% RSLogix 500 project 01. Basic_Instructions.RSS, saved by version 8.30.00.16 %
PROJECT "UNTITLED"    % processor: Bul.1763 MicroLogix 1100 Series B %

PROGRAM FILES
  LAD 2 "MAIN"  8 rungs
  LAD 3 "RTO E RES"  4 rungs
  LAD 4 "NEG E ABS"  3 rungs
  LAD 5 "RET E TND"  6 rungs
  LAD 6 "SUB RET"  6 rungs
  LAD 7 "AND, OR"  7 rungs  % And, Or, Not, Clear %
  LAD 8 "AIC E ACI"  9 rungs
  LAD 9 "AEC E AEX"  5 rungs
  LAD 10 "ACN E ASR"  5 rungs

DATA FILES
  O0 OUTPUT  4 elements
  I1 INPUT  6 elements
  S2 STATUS  66 elements
  B3 BINARY  2 elements
  T4 TIMER  2 elements
  C5 COUNTER  1 elements
  R6 CONTROL  1 elements
  N7 INTEGER  6 elements
  F8 FLOAT  1 elements
  B9 BINARY  6 elements
  ST10 STRINGS  12 elements
  N11 INTEIROS  15 elements

LADDER 2 "MAIN"
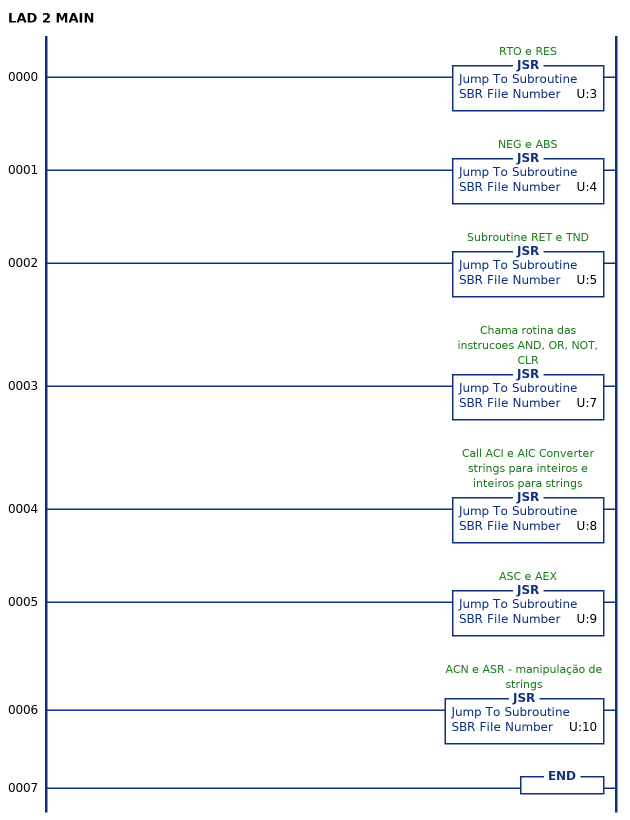
% Rung: 0 %
SOR JSR U:3 EOR
%   U:3  "RTO e RES" %
% Rung: 1 %
SOR JSR U:4 EOR
%   U:4  "NEG e ABS" %
% Rung: 2 %
SOR JSR U:5 EOR
%   U:5  "Subroutine RET e TND" %
% Rung: 3 %
SOR JSR U:7 EOR
%   U:7  "Chama rotina das instrucoes AND, OR, NOT, CLR" %
% Rung: 4 %
SOR JSR U:8 EOR
%   U:8  "Call ACI e AIC Converter strings para inteiros e inteiros para strings" %
% Rung: 5 %
SOR JSR U:9 EOR
%   U:9  "ASC e AEX" %
% Rung: 6 %
SOR JSR U:10 EOR
%   U:10  "ACN e ASR - manipulação de strings" %
% Rung: 7 %
SOR END EOR

LADDER 3 "RTO E RES"
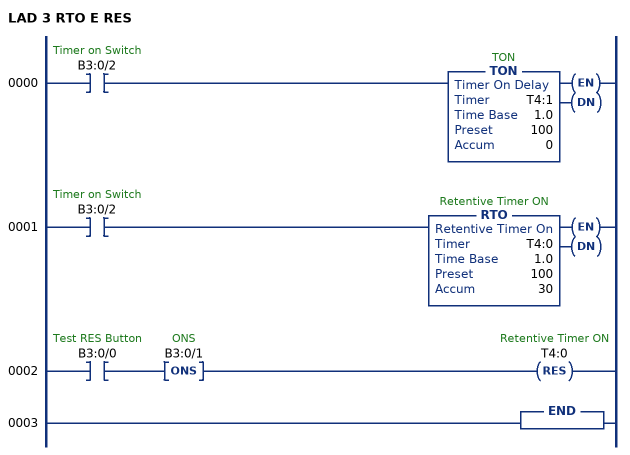
% Rung: 0 %
SOR XIC B3:0/2 TON T4:1 1.0 100 0 EOR
%   B3:0/2  "Timer on Switch" %
%   T4:1  "TON" %
% Rung: 1 %
SOR XIC B3:0/2 RTO T4:0 1.0 100 30 EOR
%   B3:0/2  "Timer on Switch" %
%   T4:0  "Retentive Timer ON" %
% Rung: 2 %
SOR XIC B3:0/0 ONS B3:0/1 RES T4:0 EOR
%   B3:0/0  "Test RES Button" %
%   B3:0/1  "ONS" %
%   T4:0  "Retentive Timer ON" %
% Rung: 3 %
SOR END EOR

LADDER 4 "NEG E ABS"
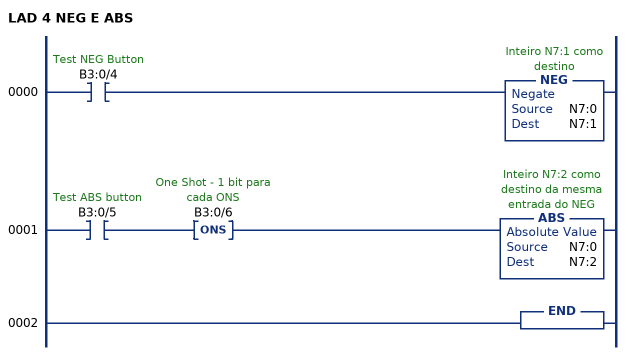
% Rung: 0 %
SOR XIC B3:0/4 NEG N7:0 N7:1 EOR
%   B3:0/4  "Test NEG Button" %
%   N7:0  "Inteiro N7:0 como entrada" %
%   N7:1  "Inteiro N7:1 como destino" %
% Rung: 1 %
SOR XIC B3:0/5 ONS B3:0/6 ABS N7:0 N7:2 EOR
%   B3:0/5  "Test ABS button" %
%   B3:0/6  "One Shot - 1 bit para cada ONS" %
%   N7:0  "Inteiro N7:0 como entrada" %
%   N7:2  "Inteiro N7:2 como destino da mesma entrada do NEG" %
% Rung: 2 %
SOR END EOR

LADDER 5 "RET E TND"
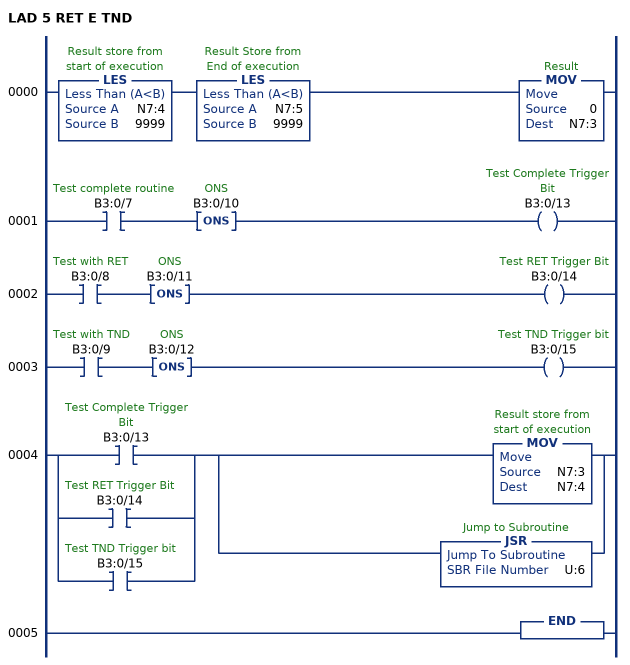
% Rung: 0 %
SOR LES N7:4 9999 LES N7:5 9999 MOV 0 N7:3 EOR
%   N7:4  "Result store from start of execution" %
%   N7:5  "Result Store from End of execution" %
%   N7:3  "Result" %
% Rung: 1 %
SOR XIC B3:0/7 ONS B3:0/10 OTE B3:0/13 EOR
%   B3:0/7  "Test complete routine" %
%   B3:0/10  "ONS" %
%   B3:0/13  "Test Complete Trigger Bit" %
% Rung: 2 %
SOR XIC B3:0/8 ONS B3:0/11 OTE B3:0/14 EOR
%   B3:0/8  "Test with RET" %
%   B3:0/11  "ONS" %
%   B3:0/14  "Test RET Trigger Bit" %
% Rung: 3 %
SOR XIC B3:0/9 ONS B3:0/12 OTE B3:0/15 EOR
%   B3:0/9  "Test with TND" %
%   B3:0/12  "ONS" %
%   B3:0/15  "Test TND Trigger bit" %
% Rung: 4 %
SOR BST XIC B3:0/13 NXB XIC B3:0/14 NXB XIC B3:0/15 BND BST MOV N7:3 N7:4 NXB JSR U:6 BND EOR
%   B3:0/13  "Test Complete Trigger Bit" %
%   B3:0/14  "Test RET Trigger Bit" %
%   B3:0/15  "Test TND Trigger bit" %
%   N7:3  "Result" %
%   N7:4  "Result store from start of execution" %
%   U:6  "Jump to Subroutine" %
% Rung: 5 %
SOR END EOR

LADDER 6 "SUB RET"
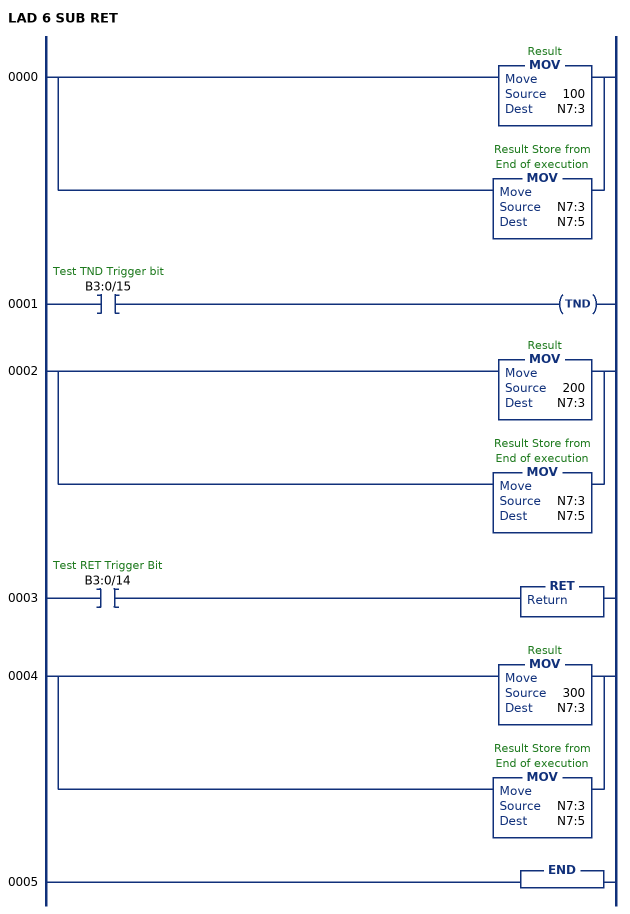
% Rung: 0 %
SOR BST MOV 100 N7:3 NXB MOV N7:3 N7:5 BND EOR
%   N7:3  "Result" %
%   N7:5  "Result Store from End of execution" %
% Rung: 1 %
SOR XIC B3:0/15 TND EOR
%   B3:0/15  "Test TND Trigger bit" %
% Rung: 2 %
SOR BST MOV 200 N7:3 NXB MOV N7:3 N7:5 BND EOR
%   N7:3  "Result" %
%   N7:5  "Result Store from End of execution" %
% Rung: 3 %
SOR XIC B3:0/14 RET EOR
%   B3:0/14  "Test RET Trigger Bit" %
% Rung: 4 %
SOR BST MOV 300 N7:3 NXB MOV N7:3 N7:5 BND EOR
%   N7:3  "Result" %
%   N7:5  "Result Store from End of execution" %
% Rung: 5 %
SOR END EOR

LADDER 7 "AND, OR"    % And, Or, Not, Clear %
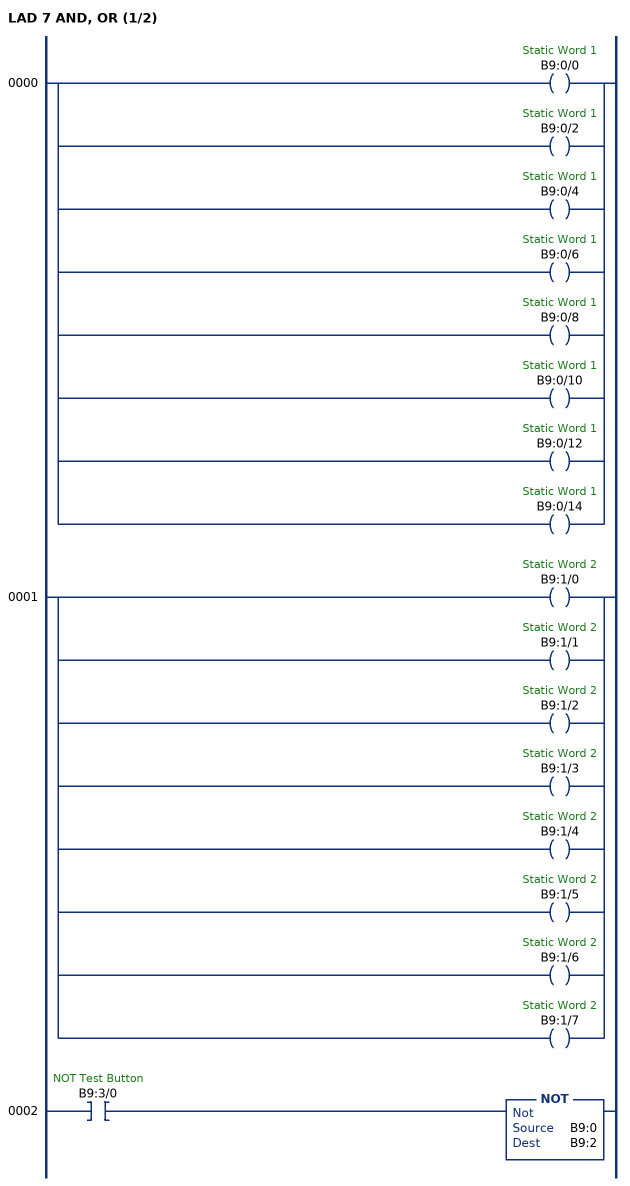
% Rung: 0 %
SOR BST OTE B9:0/0 NXB OTE B9:0/2 NXB OTE B9:0/4 NXB OTE B9:0/6 NXB OTE B9:0/8 NXB OTE B9:0/10 NXB OTE B9:0/12 NXB OTE B9:0/14 BND EOR
%   B9:0/0  "Static Word 1" %
%   B9:0/2  "Static Word 1" %
%   B9:0/4  "Static Word 1" %
%   B9:0/6  "Static Word 1" %
%   B9:0/8  "Static Word 1" %
%   B9:0/10  "Static Word 1" %
%   B9:0/12  "Static Word 1" %
%   B9:0/14  "Static Word 1" %
% Rung: 1 %
SOR BST OTE B9:1/0 NXB OTE B9:1/1 NXB OTE B9:1/2 NXB OTE B9:1/3 NXB OTE B9:1/4 NXB OTE B9:1/5 NXB OTE B9:1/6 NXB OTE B9:1/7 BND EOR
%   B9:1/0  "Static Word 2" %
%   B9:1/1  "Static Word 2" %
%   B9:1/2  "Static Word 2" %
%   B9:1/3  "Static Word 2" %
%   B9:1/4  "Static Word 2" %
%   B9:1/5  "Static Word 2" %
%   B9:1/6  "Static Word 2" %
%   B9:1/7  "Static Word 2" %
% Rung: 2 %
SOR XIC B9:3/0 NOT B9:0 B9:2 EOR
%   B9:3/0  "NOT Test Button" %
%   B9:0  "Result Word" %

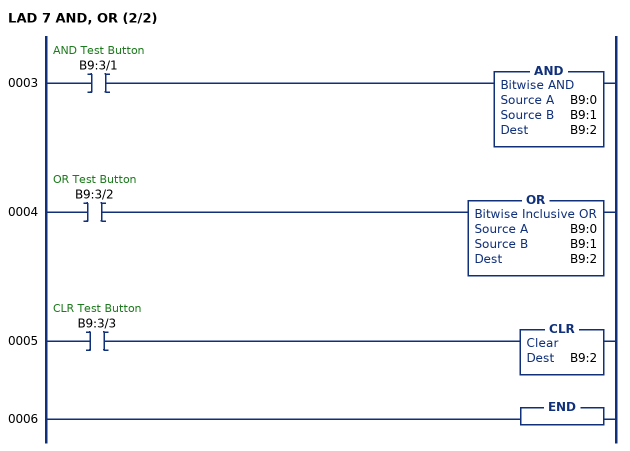
% Rung: 3 %
SOR XIC B9:3/1 AND B9:0 B9:1 B9:2 EOR
%   B9:3/1  "AND Test Button" %
%   B9:0  "Result Word" %
%   B9:1  "Result Word" %
% Rung: 4 %
SOR XIC B9:3/2 OR B9:0 B9:1 B9:2 EOR
%   B9:3/2  "OR Test Button" %
%   B9:0  "Result Word" %
%   B9:1  "Result Word" %
% Rung: 5 %
SOR XIC B9:3/3 CLR B9:2 EOR
%   B9:3/3  "CLR Test Button" %
% Rung: 6 %
SOR END EOR

LADDER 8 "AIC E ACI"
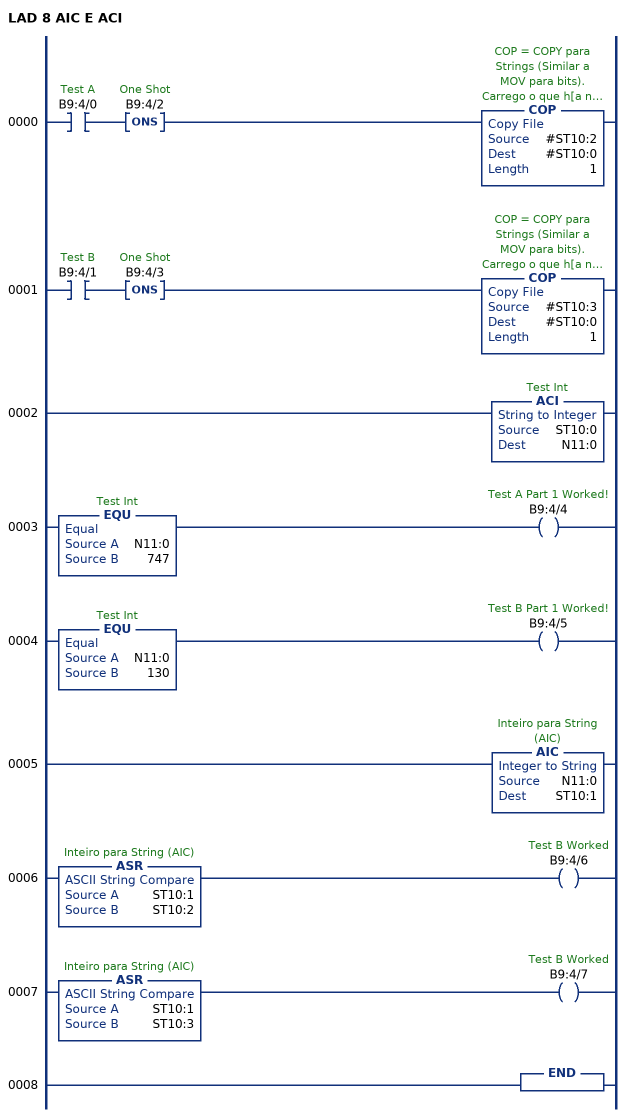
% Rung: 0 %
SOR XIC B9:4/0 ONS B9:4/2 COP #ST10:2 #ST10:0 1 EOR
%   B9:4/0  "Test A" %
%   B9:4/2  "One Shot" %
%   ST10:2  "COP = COPY para Strings. Carrego o valor da String ST9:2 para ST9:0" %
%   ST10:0  "COP = COPY para Strings (Similar a MOV para bits). Carrego o que h[a na String ST10:2 0" %
% Rung: 1 %
SOR XIC B9:4/1 ONS B9:4/3 COP #ST10:3 #ST10:0 1 EOR
%   B9:4/1  "Test B" %
%   B9:4/3  "One Shot" %
%   ST10:3  "Test String" %
%   ST10:0  "COP = COPY para Strings (Similar a MOV para bits). Carrego o que h[a na String ST10:2 0" %
% Rung: 2 %
SOR ACI ST10:0 N11:0 EOR
%   ST10:0  "COP = COPY para Strings (Similar a MOV para bits). Carrego o que h[a na String ST10:2 0" %
%   N11:0  "Test Int" %
% Rung: 3 %
SOR EQU N11:0 747 OTE B9:4/4 EOR
%   N11:0  "Test Int" %
%   B9:4/4  "Test A Part 1 Worked!" %
% Rung: 4 %
SOR EQU N11:0 130 OTE B9:4/5 EOR
%   N11:0  "Test Int" %
%   B9:4/5  "Test B Part 1 Worked!" %
% Rung: 5 %
SOR AIC N11:0 ST10:1 EOR
%   N11:0  "Test Int" %
%   ST10:1  "Inteiro para String (AIC)" %
% Rung: 6 %
SOR ASR ST10:1 ST10:2 OTE B9:4/6 EOR
%   ST10:1  "Inteiro para String (AIC)" %
%   ST10:2  "COP = COPY para Strings. Carrego o valor da String ST9:2 para ST9:0" %
%   B9:4/6  "Test B Worked" %
% Rung: 7 %
SOR ASR ST10:1 ST10:3 OTE B9:4/7 EOR
%   ST10:1  "Inteiro para String (AIC)" %
%   ST10:3  "Test String" %
%   B9:4/7  "Test B Worked" %
% Rung: 8 %
SOR END EOR

LADDER 9 "AEC E AEX"
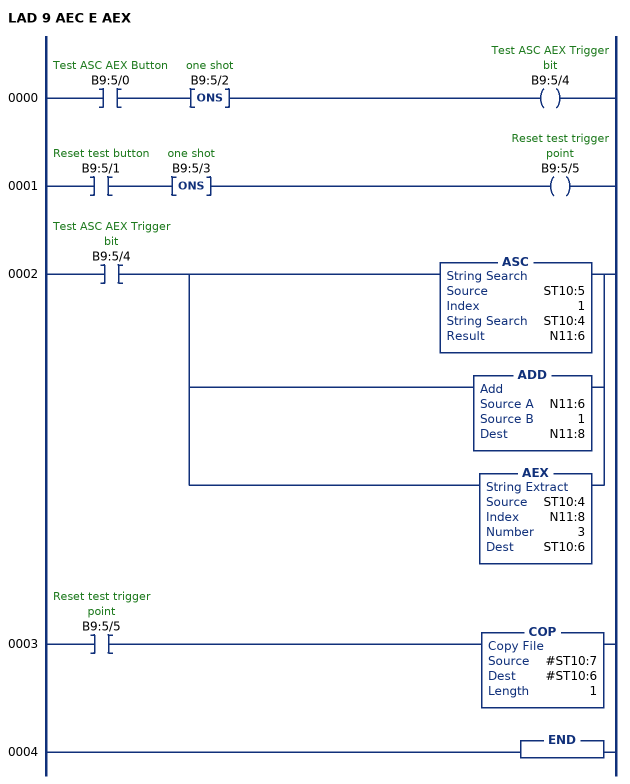
% Rung: 0 %
SOR XIC B9:5/0 ONS B9:5/2 OTE B9:5/4 EOR
%   B9:5/0  "Test ASC AEX Button" %
%   B9:5/2  "one shot" %
%   B9:5/4  "Test ASC AEX Trigger bit" %
% Rung: 1 %
SOR XIC B9:5/1 ONS B9:5/3 OTE B9:5/5 EOR
%   B9:5/1  "Reset test button" %
%   B9:5/3  "one shot" %
%   B9:5/5  "Reset test trigger point" %
% Rung: 2 %
SOR XIC B9:5/4 BST ASC ST10:5 1 ST10:4 N11:6 NXB ADD N11:6 1 N11:8 NXB AEX ST10:4 N11:8 3 ST10:6 BND EOR
%   B9:5/4  "Test ASC AEX Trigger bit" %
% Rung: 3 %
SOR XIC B9:5/5 COP #ST10:7 #ST10:6 1 EOR
%   B9:5/5  "Reset test trigger point" %
% Rung: 4 %
SOR END EOR

LADDER 10 "ACN E ASR"
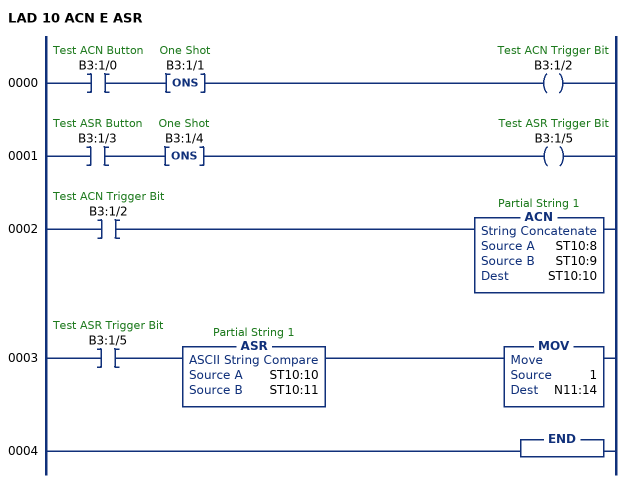
% Rung: 0 %
SOR XIC B3:1/0 ONS B3:1/1 OTE B3:1/2 EOR
%   B3:1/0  "Test ACN Button" %
%   B3:1/1  "One Shot" %
%   B3:1/2  "Test ACN Trigger Bit" %
% Rung: 1 %
SOR XIC B3:1/3 ONS B3:1/4 OTE B3:1/5 EOR
%   B3:1/3  "Test ASR Button" %
%   B3:1/4  "One Shot" %
%   B3:1/5  "Test ASR Trigger Bit" %
% Rung: 2 %
SOR XIC B3:1/2 ACN ST10:8 ST10:9 ST10:10 EOR
%   B3:1/2  "Test ACN Trigger Bit" %
%   ST10:9  "Partial String 1" %
%   ST10:10  "Partial String 1" %
% Rung: 3 %
SOR XIC B3:1/5 ASR ST10:10 ST10:11 MOV 1 N11:14 EOR
%   B3:1/5  "Test ASR Trigger Bit" %
%   ST10:10  "Partial String 1" %
% Rung: 4 %
SOR END EOR

OTHER DOCUMENTED ADDRESSES
  B9:0/1  "Static Word 1"
  N11:2  "Target Start index"

DATA TABLE (non-zero values as saved)
DATA B3
% B3:0 % 0X0003 0X0003
DATA T4
% .PRE .ACC %
% T4:0 % 100 30
% T4:1 % 100 0
DATA N7
% N7:0 % 25 -25 25 0 0 100
DATA B9
% B9:0 % 0X5555 0X00FF 0X0000 0X0008 0X0005 0X0005
DATA ST10
% ST10:0 % "dash^&-plc$stuff"
% ST10:1 % "0"
% ST10:4 % "dash^&-plc$stuff"
% ST10:5 % "-"
% ST10:6 % "plc"
% ST10:8 % "TEST"
% ST10:9 % "STRING"
% ST10:10 % "TESTSTRING"
% ST10:11 % "TESTSTRING"
DATA N11
% N11:0 % 0 0 1 0 0 0 8 0 9 0
